FUNCTION_BLOCK FB_PCMStorage
VAR_INPUT
END_VAR
VAR_OUTPUT
	{attribute 'OPC.UA.DA' := '1'}
	localState : ST_PCMStorageState;
END_VAR
VAR
	//temperature sensors
	TemperatureSensor : FB_TemperatureSensor_KL3214;
	
	//Temperature
	Temperature: REAL;
	
	// SOC-Value
	SOC_per : REAL; 
	SOC_abs : REAL; 
	
END_VAR

//temperature sensors
TemperatureSensor();
TemperatureSensor.GetState_AI();

Temperature := TemperatureSensor.fTemperature;

CalcSOC(
    Temperature := Temperature, 
    SOC_per => localState.SOCValuePercentage, 
    SOC_abs => localState.SOCValueAbsolute
);

localState.SOCValuePercentage := SOC_per; 
localState.SOCValueAbsolute := SOC_abs; 
localState.TemperatureSensor := Temperature;

METHOD CalcSOC : REAL
VAR_INPUT
	Temperature: REAL;
END_VAR
VAR_OUTPUT
	SOC_per : REAL;
	SOC_abs : REAL;
END_VAR
//derivation and parameter from jonas wendts dissertation
SOC_per := (0.11822542*EXPT(Temperature, 4)-7.4519133*EXPT(Temperature, 3)+174.94045*EXPT(Temperature, 2)-1822.0902*Temperature+7168.3066);

IF SOC_per > 100 THEN
	SOC_per := 100;
ELSIF SOC_per > 100 THEN
	SOC_per := 0; 
END_IF

SOC_abs := (SOC_per/100)*20.43;
END_METHOD

END_FUNCTION_BLOCK

(* stored: Version 1.1.0.1, ProductVersion 3.1.4024.10
   POU FB_PCMStorage: Id {069b991a-1373-4b42-afea-bf8744e0dec1}, SpecialFunc None
   Method CalcSOC: Id {1ae693ec-0905-444f-a924-e5322946a7f4} *)
